{attribute addProperty BoxType "EK1100-0000-0018"}
{attribute addProperty Id "Beckhoff_EJ1xxxEK1122Beckhoff_EJ1xxxEK1122_5D41058A11314.125A_0004_EJ1008_0000_0017EJ1008_772BB4148210.25A_0005_EJ1128_0000_0016EJ1128_772BB4148210.25A_0006_EJ1809_0000_0017EJ1809_248EAA3414618.25A_0007_EJ1819_0000_0017EJ1819_248EAA3414618.25A_0008_EJ1859_0000_0017EJ1859_538B459D14618.25A_0009_EJ1889_0000_0017EJ1889_248EAA3414618.25A_0003_EJ1122_0000_0016EJ1122_179A0949162"}
{attribute addProperty CRC "3125669324"}
{attribute addProperty SizeInBites "877"}
{attribute addProperty SizeInBytes "109.625"}
TYPE Beckhoff_EJ1xxx_BA4DEDCC EXTENDS EK1100_179A0949 :
STRUCT
	{attribute addProperty Name "Beckhoff_EJ1xxxEK1122"}
	Beckhoff_EJ1xxxEK1122 : Beckhoff_EJ1xxxEK1122_5D41058A;
	{attribute addProperty Name "A_0004_EJ1008_0000_0017"}
	A_0004_EJ1008_0000_0017 : EJ1008_772BB414;
	{attribute addProperty Name "A_0005_EJ1128_0000_0016"}
	A_0005_EJ1128_0000_0016 : EJ1128_772BB414;
	{attribute addProperty Name "A_0006_EJ1809_0000_0017"}
	A_0006_EJ1809_0000_0017 : EJ1809_248EAA34;
	{attribute addProperty Name "A_0007_EJ1819_0000_0017"}
	A_0007_EJ1819_0000_0017 : EJ1819_248EAA34;
	{attribute addProperty Name "A_0008_EJ1859_0000_0017"}
	A_0008_EJ1859_0000_0017 : EJ1859_538B459D;
	{attribute addProperty Name "A_0009_EJ1889_0000_0017"}
	A_0009_EJ1889_0000_0017 : EJ1889_248EAA34;
	{attribute addProperty Name "A_0003_EJ1122_0000_0016"}
	A_0003_EJ1122_0000_0016 : EJ1122_179A0949;
END_STRUCT
END_TYPE

(* stored: Version 1.2.0.0, ProductVersion 3.1.4024.9
   DUT Beckhoff_EJ1xxx_BA4DEDCC: Id {99ccd103-12b5-4c0c-a100-04f15ed08c1b} *)
